// TwinCAT 3 PLC project mobject_commands
// Title: mobject-commands
// Company: mobject
// Author: mobject dev team
// ProjectVersion: 0.2.0
// ProgramVersion: 3.1.4024.0
// libraries:
//   Tc2_System, * (Beckhoff Automation GmbH)
//   mobject-disposable,1.1.1,mobject
// project tree:
//   AsyncCommand/Interface/ I_AsyncCommand.TcIO
//   AsyncCommand/ AsyncCommand.TcPOU
//   AsyncCommand/Runners/ SingleAsyncCommandRunner.TcPOU
//   Command/Interface/ I_Command.TcIO
//   _Internal/AsyncCommandStateMachine/ AsyncCommandStateMachine.TcPOU, I_AsyncCommandStateControl.TcIO

// ---- AsyncCommand/Interface/I_AsyncCommand.TcIO
INTERFACE I_AsyncCommand extends I_Command

METHOD PUBLIC Abort
VAR_INPUT
END_VAR
END_METHOD

PROPERTY PUBLIC Busy : BOOL
GET
END_GET
END_PROPERTY

METHOD PUBLIC CyclicCall
VAR_INPUT
END_VAR
END_METHOD

PROPERTY PUBLIC Done : BOOL
GET
END_GET
END_PROPERTY

PROPERTY PUBLIC Error : BOOL
GET
END_GET
END_PROPERTY

PROPERTY PUBLIC ErrorId : UDINT
GET
END_GET
END_PROPERTY

END_INTERFACE

// ---- Command/Interface/I_Command.TcIO
INTERFACE I_Command EXTENDS I_Disposable

METHOD Execute
VAR_INPUT
END_VAR
END_METHOD

END_INTERFACE

// ---- _Internal/AsyncCommandStateMachine/I_AsyncCommandStateControl.TcIO
INTERFACE I_AsyncCommandStateControl

METHOD PUBLIC Error
VAR_INPUT
	ErrorId : UDINT;
END_VAR
END_METHOD

METHOD PUBLIC Next
VAR_INPUT
END_VAR
END_METHOD

END_INTERFACE

// ---- AsyncCommand/AsyncCommand.TcPOU
{attribute 'linkalways'} 
{attribute 'no_explicit_call' := 'This FB is a CLASS and must be accessed using methods or properties'}
{attribute 'enable_dynamic_creation'}
FUNCTION_BLOCK AsyncCommand EXTENDS Disposable IMPLEMENTS I_AsyncCommand
VAR
	stateMachine : AsyncCommandStateMachine;
END_VAR

METHOD PUBLIC Abort
VAR_INPUT
END_VAR
stateMachine.Abort();
END_METHOD

PROPERTY PUBLIC Busy : BOOL
GET
IF stateMachine.IsAborted THEN
	RETURN;
END_IF

IF stateMachine.IsCompleted THEN
	RETURN;
END_IF

IF stateMachine.IsErrored THEN
	RETURN;
END_IF

IF stateMachine.IsIdle THEN
	RETURN;
END_IF

Busy := TRUE;
END_GET
END_PROPERTY

METHOD PUBLIC CyclicCall
VAR_INPUT
END_VAR
IF stateMachine.IsIdle THEN
	OnIdle();
END_IF

IF stateMachine.IsInitializing THEN
	OnInitializing(stateMachine);
END_IF

IF stateMachine.IsExecuting THEN
	OnExecuting(stateMachine);
END_IF

IF stateMachine.IsCompleting THEN
	OnCompleting(stateMachine);
END_IF

IF stateMachine.IsCompleted THEN
	OnCompleted();
END_IF

IF stateMachine.IsAborting THEN
	OnAborting(stateMachine);
END_IF

IF stateMachine.IsAborted THEN
	OnAborted();
END_IF

IF stateMachine.IsErrored THEN
	OnErrored();
END_IF
END_METHOD

PROPERTY PUBLIC Done : BOOL
GET
Done := stateMachine.IsCompleted;
END_GET
END_PROPERTY

PROPERTY PUBLIC Error : BOOL
GET
Error := stateMachine.IsErrored;
END_GET
END_PROPERTY

PROPERTY PUBLIC ErrorId : UDINT
GET
ErrorId := stateMachine.ErrorId;
END_GET
END_PROPERTY

METHOD PUBLIC Execute
VAR_INPUT
END_VAR
stateMachine.Execute();
END_METHOD

METHOD PROTECTED OnAborted
VAR_INPUT
END_VAR
END_METHOD

METHOD PROTECTED OnAborting
VAR_INPUT
	StateControl : I_AsyncCommandStateControl;
END_VAR
// default behaviour is to go to next state
// you can override this method to implement your own completing control code.
// just call StateControl.Next() when your code is completed.  

StateControl.Next();
END_METHOD

METHOD PROTECTED OnCompleted : BOOL
VAR_INPUT
END_VAR
END_METHOD

METHOD PROTECTED OnCompleting
VAR_INPUT
	StateControl : I_AsyncCommandStateControl;
END_VAR
// default behaviour is to go to next state
// you can override this method to implement your own completing control code.
// just call StateControl.Next() when your code is completed.  

StateControl.Next();
END_METHOD

METHOD PROTECTED OnErrored
VAR_INPUT
END_VAR
END_METHOD

METHOD PROTECTED OnExecuting
VAR_INPUT
	StateControl : I_AsyncCommandStateControl;
END_VAR
// default behaviour is to go to next state
// you can override this method to implement your own executing control code.
// just call StateControl.Next() when your code is completed.  

StateControl.Next();
END_METHOD

METHOD PROTECTED OnIdle
VAR_INPUT
END_VAR
END_METHOD

METHOD PROTECTED OnInitializing
VAR_INPUT
	StateControl : I_AsyncCommandStateControl;
END_VAR
// default behaviour is to go to next state
// you can override this method to implement your own initializing control code.
// just call StateControl.Next() when your code is completed.  

StateControl.Next();
END_METHOD

END_FUNCTION_BLOCK

// ---- _Internal/AsyncCommandStateMachine/AsyncCommandStateMachine.TcPOU
{attribute 'linkalways'} 
{attribute 'no_explicit_call' := 'This FB is a CLASS and must be accessed using methods or properties'}
{attribute 'enable_dynamic_creation'}
FUNCTION_BLOCK AsyncCommandStateMachine IMPLEMENTS I_AsyncCommandStateControl
VAR
	state : (IDLE, INITIALIZING, EXECUTING, COMPLETING, COMPLETED, ABORTING, ABORTED, ERRORED);
	_errorId : UDINT;
END_VAR

METHOD PUBLIC Abort
VAR_INPUT
END_VAR
CASE state OF
	IDLE : RETURN;
	ABORTING : RETURN;
	COMPLETED : RETURN;
	ABORTED : RETURN;
	ERRORED : RETURN;
END_CASE

state := ABORTING;
END_METHOD

METHOD PUBLIC Error
VAR_INPUT
	ErrorId : UDINT;
END_VAR
CASE state OF
	IDLE : RETURN;
	COMPLETED : RETURN;
	ABORTED : RETURN;
	ERRORED : RETURN;
END_CASE

_errorId := ErrorId;
state := ERRORED;
END_METHOD

{attribute 'monitoring' := 'call'}
PROPERTY PUBLIC ErrorId : UDINT
GET
ErrorID := _errorId;
END_GET
END_PROPERTY

METHOD PUBLIC Execute
VAR_INPUT
END_VAR
CASE state OF
	INITIALIZING : RETURN;
	EXECUTING : RETURN;
	COMPLETING : RETURN;
	ABORTING : RETURN;
END_CASE

_errorId := 0;
state := INITIALIZING;
END_METHOD

{attribute 'monitoring' := 'call'}
PROPERTY PUBLIC IsAborted : BOOL
GET
IsAborted := state = ABORTED;
END_GET
END_PROPERTY

{attribute 'monitoring' := 'call'}
PROPERTY PUBLIC IsAborting : BOOL
GET
IsAborting := state = ABORTING;
END_GET
END_PROPERTY

{attribute 'monitoring' := 'call'}
PROPERTY PUBLIC IsCompleted : BOOL
GET
IsCompleted := state = COMPLETED;
END_GET
END_PROPERTY

{attribute 'monitoring' := 'call'}
PROPERTY PUBLIC IsCompleting : BOOL
GET
IsCompleting := state = COMPLETING;
END_GET
END_PROPERTY

{attribute 'monitoring' := 'call'}
PROPERTY PUBLIC IsErrored : BOOL
GET
IsErrored := state = ERRORED;
END_GET
END_PROPERTY

{attribute 'monitoring' := 'call'}
PROPERTY PUBLIC IsExecuting : BOOL
GET
IsExecuting := state = EXECUTING;
END_GET
END_PROPERTY

{attribute 'monitoring' := 'call'}
PROPERTY PUBLIC IsIdle : BOOL
GET
IsIdle:= state = IDLE;
END_GET
END_PROPERTY

{attribute 'monitoring' := 'call'}
PROPERTY PUBLIC IsInitializing : BOOL
GET
IsInitializing := state = INITIALIZING;
END_GET
END_PROPERTY

METHOD PUBLIC Next
VAR_INPUT
END_VAR
CASE state OF
	IDLE : RETURN;
	INITIALIZING : StateComplete_Initializing();
	EXECUTING : StateComplete_Executing();
	COMPLETING : StateComplete_Completing();
	COMPLETED : RETURN;
	ABORTING : StateComplete_Aborting();
	ABORTED : RETURN;
	ERRORED : RETURN;
END_CASE
END_METHOD

METHOD PRIVATE StateComplete_Aborting
VAR_INPUT
END_VAR
state := ABORTED;
END_METHOD

METHOD PRIVATE StateComplete_Completing
VAR_INPUT
END_VAR
state := COMPLETED;
END_METHOD

METHOD PRIVATE StateComplete_Executing
VAR_INPUT
END_VAR
state := COMPLETING;
END_METHOD

METHOD PRIVATE StateComplete_Initializing
VAR_INPUT
END_VAR
state := EXECUTING;
END_METHOD

END_FUNCTION_BLOCK

// ---- AsyncCommand/Runners/SingleAsyncCommandRunner.TcPOU
{attribute 'linkalways'} 
{attribute 'no_explicit_call' := 'This FB is a CLASS and must be accessed using methods or properties'}
{attribute 'enable_dynamic_creation'}
FUNCTION_BLOCK SingleAsyncCommandRunner
VAR
	currentCommand : I_AsyncCommand;
	replacementCommand : I_AsyncCommand;
END_VAR

PROPERTY PUBLIC Busy : BOOL
GET
IF currentCommand = 0 THEN
	RETURN;
END_IF

Busy := currentCommand.Busy;
END_GET
END_PROPERTY

METHOD PUBLIC CyclicCall
VAR_INPUT
END_VAR
IF currentCommand <> 0 AND_THEN currentCommand.Busy THEN
	currentCommand.CyclicCall();
	RETURN;
END_IF

IF replacementCommand <> 0 THEN
	currentCommand := replacementCommand;
	replacementCommand := 0;
	currentCommand.Execute();
END_IF
END_METHOD

PROPERTY Done : BOOL
GET
IF currentCommand = 0 THEN
	RETURN;
END_IF

Done := currentCommand.Done;
END_GET
END_PROPERTY

PROPERTY Error : BOOL
GET
IF currentCommand = 0 THEN
	RETURN;
END_IF

Error := currentCommand.Error;
END_GET
END_PROPERTY

PROPERTY PUBLIC ErrorId : UDINT
GET
IF currentCommand = 0 THEN
	RETURN;
END_IF

ErrorId := currentCommand.ErrorId;
END_GET
END_PROPERTY

METHOD ExecuteCommand
VAR_INPUT
	Command : I_AsyncCommand;
END_VAR
IF currentCommand = 0 THEN
	currentCommand := Command;
	currentCommand.Execute();
	RETURN;
END_IF

currentCommand.Abort();
replacementCommand := Command;
END_METHOD

END_FUNCTION_BLOCK
